RESOURCE_TYPE DE2_115
  (* Standard: 61499-2 *)
  (* Version 0.1, 2016-00-08, hpea485, UOA *)
  FBS
    conveyor : Conveyor_SIFB;
    globals : Globals_SIFB;
    boxdropper : BoxDropper_SIFB;
  END_FBS
  EVENT_CONNECTIONS
    globals.global_run_changed TO conveyor.conveyor_run_changed;
    globals.global_run_changed TO boxdropper.box_dropper_run_changed;
  END_CONNECTIONS
  DATA_CONNECTIONS
    globals.global_run_infinite TO conveyor.conveyor_run;
    globals.global_run_infinite TO boxdropper.box_dropper_run;
  END_CONNECTIONS
END_RESOURCE_TYPE
